# EPICS substitutions: example/exampleApp/Db/example.substitutions
file mettlerToledo.template
{
pattern {P, PORT, ADDR}
        {mkp:SE:Scale, MT1, 0}
}
